// TIA Portal V19 export
TYPE "lexchangetray_typeUnEmn_toConstraintWorkstationReq"
// Type: Bool
// stored: Access Published
   STRUCT
      transferEnable : Bool;   // 请求转移
      unConstraint : Bool;
      Constraint : Bool;
   END_STRUCT;
END_TYPE
